PROGRAM master
VAR
	axis				: AXIS_REF;
	
	mcPower				: MC_Power;
	shouldPowerOn		: BOOL;
	isMotorReady		: BOOL;
	
	mcSetPosition		: MC_SetPosition;
	shouldSetZero		: BOOL;
	
	mcJog				: MC_Jog;
	shouldJog			: BOOL;
	jogDirection		: BOOL;
	
	mcMoveRelative		: MC_MoveRelative;
	shouldMoveRel		: BOOL;
	
	mcStop				: MC_Stop;
	shouldStop			: BOOL;
	
	mcReset				: MC_Reset;
	shouldReset			: BOOL;
	
	mcHome				: MC_Home;
	shouldGoHome		: BOOL;
	homeTrigger			: BOOL;
END_VAR

METHOD checkGoHome : BOOL
VAR_INPUT
END_VAR
mcHome(
	Axis:= axis, 
	Execute:= shouldGoHome, 
	Position:= 0, 
	bCalibrationCam:= homeTrigger
);
END_METHOD

METHOD checkMoving : BOOL
VAR_STAT
END_VAR
IF isMotorReady THEN
	IF shouldJog THEN
		IF jogDirection THEN
		mcJog(
			Axis:= axis, 
			JogForward:= TRUE, 
			JogBackwards:= FALSE,
			Velocity:= 50);
		ELSE
			mcJog(
				Axis:= axis, 
				JogForward:= FALSE, 
				JogBackwards:= TRUE,
				Velocity:= 50);
		END_IF
	END_IF
END_IF
END_METHOD

METHOD checkPower : BOOL
VAR_INPUT
END_VAR
VAR
END_VAR
mcPower(
	Axis:= axis, 
	Enable:= shouldPowerOn, 
	Enable_Positive:= TRUE, 
	Enable_Negative:= TRUE,
	Status=> isMotorReady
);
END_METHOD

METHOD checkRelMove : BOOL
VAR_STAT
END_VAR
IF isMotorReady THEN
	mcMoveRelative(
		Axis:= axis, 
		Execute:= shouldMoveRel, 
		Distance:= 2000, 
		Velocity:= 50);
END_IF;
END_METHOD

METHOD checkReset : BOOL
IF isMotorReady THEN
	mcReset(
		Axis:= axis, 
		Execute:= shouldReset);
END_IF
END_METHOD

ACTION checkSetPoint:
mcSetPosition(
	Axis:= axis, 
	Execute:= shouldSetZero,
	Position := 0);
END_ACTION

METHOD checkStop : BOOL
VAR

END_VAR
IF isMotorReady THEN
	mcStop(
		Axis:= axis, 
		Execute:= shouldStop);
END_IF
END_METHOD

ACTION dummyAction:

END_ACTION

END_PROGRAM

(* stored: Version 1.1.0.1, ProductVersion 3.1.4024.4
   POU master: Id {51f8bfd8-5336-424e-9d39-0ed2ef8b99b5}, SpecialFunc None
   Method checkGoHome: Id {7375619a-1d8c-4819-9be5-1e8c5db522ae}
   Method checkMoving: Id {09805a7c-6bc1-4dd6-8c96-108ff965a2e0}
   Method checkPower: Id {c64668b3-b8f3-4c8c-9e2d-b6feb4467932}
   Method checkRelMove: Id {5a093290-3d42-43f3-afd9-4ef4314b7508}
   Method checkReset: Id {524a7df7-b01b-404f-8b9e-670d73e37929}
   Action checkSetPoint: Id {3147e69a-6538-4ecd-b3b7-7219cbda6e48}
   Method checkStop: Id {59d6d916-623b-4e33-a0e3-1cfdd666254e}
   Action dummyAction: Id {8e7a3a76-47ac-4d3e-90de-e71277f386ea} *)
